// TIA Portal V16 export
// export: Created 2024-12-03T15:41:45.4636879Z, ExportSetting WithReadOnly, DisplayName Totally Integrated Automation Portal, DisplayVersion V16 Update 6, DisplayName TIA Portal Version Control Interface, DisplayVersion V16 Update 2, DisplayName TIA Portal Openness, DisplayVersion V16 Update 6, DisplayName TIA Portal Teamcenter Gateway, DisplayVersion V16, DisplayName SINAMICS Startdrive Advanced, DisplayVersion V16 Update 5, DisplayName SINAMICS Startdrive G130, G150, S120, S150, SINAMICS MV, S210, DisplayVersion V16 Update 5, DisplayName SINAMICS Startdrive G110M, G120, G120C, G120D, G120P, G115D, DisplayVersion V16 Update 5, DisplayName STEP 7 Professional, DisplayVersion V16 Update 6, DisplayName STEP 7 Safety, DisplayVersion V16, DisplayName WinCC Advanced / Unified PC, DisplayVersion V16 Update 6
TYPE "GXXX_EXTENSION_INPUT_UDT"
// stored: CreationDate 2022-02-10T10:30:20.6863124Z, InterfaceModifiedDate 2021-08-10T11:20:06.8217946Z, IsConsistent true, LibraryConformanceStatus The object is library-conformant., ModifiedDate 2021-08-10T11:20:06.8217946Z
   STRUCT
      DigitalInputState : Struct
         di_24 : Bool;
         di_25 : Bool;
         spare_1 : Bool;
         spare_2 : Bool;
         spare_3 : Bool;
         spare_4 : Bool;
         spare_5 : Bool;
         spare_6 : Bool;
         spare_7 : Byte;
         spare_8 : Byte;
         di_0 : Bool;
         di_1 : Bool;
         di_2 : Bool;
         di_3 : Bool;
      END_STRUCT;
   END_STRUCT;
END_TYPE
